// TIA Portal project "TemperatureingangNormieren" (V14)

(* hardware
DEVICE "S7-1200-Station_1"  S7-1200 Station
   slot 0: "Baugruppenträger_0"  S7-1200 Rack  Rack  V1.0
   slot 1: "PLC_1"  CPU 1214C DC/DC/DC  6ES7 214-1AG40-0XB0  V4.2
   slot 3: "AQ 1x12BIT_1"  AQ1 signal board  6ES7 232-4HA30-0XB0  V1.0
*)

// ===== PLC "PLC_1"  CPU 1214C DC/DC/DC =====

VAR_GLOBAL   // PLC tag table "Standard-Variablentabelle"
   "System_Byte" AT %MB100 : Byte;
   "FirstScan" AT %M100.0 : Bool;
   "DiagStatusUpdate" AT %M100.1 : Bool;
   "AlwaysTRUE" AT %M100.2 : Bool;
   "AlwaysFALSE" AT %M100.3 : Bool;
   "Clock_Byte" AT %MB110 : Byte;
   "Clock_10Hz" AT %M110.0 : Bool;
   "Clock_5Hz" AT %M110.1 : Bool;
   "Clock_2.5Hz" AT %M110.2 : Bool;
   "Clock_2Hz" AT %M110.3 : Bool;
   "Clock_1.25Hz" AT %M110.4 : Bool;
   "Clock_1Hz" AT %M110.5 : Bool;
   "Clock_0.625Hz" AT %M110.6 : Bool;
   "Clock_0.5Hz" AT %M110.7 : Bool;
   "iAnalogEingang1" AT %IW64 : Int;
   "iAnalogEingang2" AT %IW66 : Int;
   "iAnalogAusgang" AT %QW80 : Int;
   "AlleAusgänge" AT %QW0 : Word;
END_VAR

DATA_BLOCK "fbTemperaturEingangNormieren_DB"   // DB1
{ S7_Optimized_Access := 'TRUE' }
VERSION : 0.1
// stored: InstanceOfName fbTemperaturEingangNormieren
"fbTemperaturEingangNormieren"
BEGIN
END_DATA_BLOCK

FUNCTION_BLOCK "fbTemperaturEingangNormieren"   // FB1, LAD
{ S7_Optimized_Access := 'TRUE' }
VERSION : 0.1
   VAR_INPUT
      iAnalogEingang : Int;   // Analogeingang (+/- 32767)
      rMinWarnung : Real;   // Warnung - unteres Limit in °C
      rMaxWarnugn : Real;   // Warnung - oberes Limit in °C
      rMinStoerung : Real;   // Störung - unteres Limit in °C
      rMaxStoerung : Real;   // Störung - oberes Limit in °C
      rHysterese : Real;   // Hysterese in °C
      iX0 : Int;   // Punkt 0 - Analogeingang
      iX1 : Int;   // Punkt 1 - Analogeingang
      rY0 : Real;   // Punkt 0 - Temperatur
      rY1 : Real;   // Punkt 1 - Temperatur
   END_VAR
   VAR_OUTPUT
      rTemperatur : Real;   // Temperatur in °C
      xMinWarnung : Bool;   // Warnung - unteres Limit
      xMaxWarnung : Bool;   // Warnung - oberes Limit
      xMinStoerung : Bool;   // Störung - unteres Limit
      xMaxStoerung : Bool;   // Störung - oberes Limit
   END_VAR
BEGIN
END_FUNCTION_BLOCK

FUNCTION "fcAnalogeingang" : Void   // FC1, LAD
{ S7_Optimized_Access := 'TRUE' }
VERSION : 0.1
BEGIN

REGION Network 1
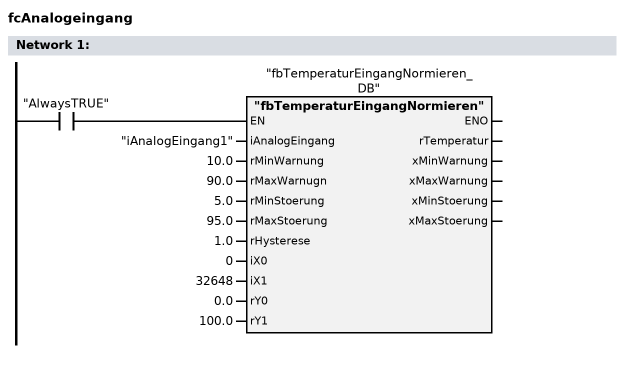
   RUNG wire#powerrail
      Contact( "AlwaysTRUE" )
      "fbTemperaturEingangNormieren_DB"(iAnalogEingang := "iAnalogEingang1", rMinWarnung := 10.0, rMaxWarnugn := 90.0, rMinStoerung := 5.0, rMaxStoerung := 95.0, rHysterese := 1.0, iX0 := 0, iX1 := 32648, rY0 := 0.0, rY1 := 100.0, rTemperatur =>, xMinWarnung =>, xMaxWarnung =>, xMinStoerung =>, xMaxStoerung =>)
   END_RUNG
   // the same network as SCL:
   IF "AlwaysTRUE" THEN
       "fbTemperaturEingangNormieren_DB"(iAnalogEingang := "iAnalogEingang1",   // "fbTemperaturEingangNormieren"
                               rMinWarnung := 10.0,
                               rMaxWarnugn := 90.0,
                               rMinStoerung := 5.0,
                               rMaxStoerung := 95.0,
                               rHysterese := 1.0,
                               iX0 := 0,
                               iX1 := 32648,
                               rY0 := 0.0,
                               rY1 := 100.0);
   END_IF;
END_REGION
END_FUNCTION

ORGANIZATION_BLOCK "Main"   // OB1, LAD, ProgramCycle
TITLE = "Main Program Sweep (Cycle)"
{ S7_Optimized_Access := 'TRUE' }
VERSION : 0.1
   VAR_INPUT
      Initial_Call : Bool;   // Initial call of this OB
      Remanence : Bool;   // =True, if remanent data are available
   END_VAR
BEGIN

REGION Network 1
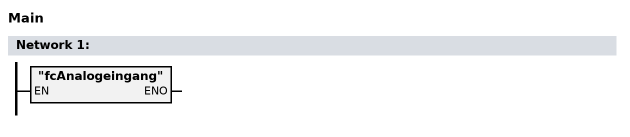
   RUNG wire#powerrail
      "fcAnalogeingang"()
   END_RUNG
   // the same network as SCL:
   "fcAnalogeingang"();
END_REGION
END_ORGANIZATION_BLOCK

ORGANIZATION_BLOCK "Startup"   // OB100, SCL, Startup
TITLE = "Complete Restart"
{ S7_Optimized_Access := 'TRUE' }
VERSION : 0.1
   VAR_INPUT
      LostRetentive : Bool;   // True if retentive data are lost
      LostRTC : Bool;   // True if date and time are lost
   END_VAR
BEGIN
   "AlleAusgänge" := 16#0000;
END_ORGANIZATION_BLOCK